{attribute 'qualified_only'}
{attribute 'strict'}
TYPE E_DALIBridgeCommand :
(
	idle,
	directArcPowerControl,
	queryActualLevel,
	queryStatus,
	setEventScheme,
	queryEventScheme,
	setEventFilter,
	queryEventFilter,
	identifyDevice102,
	identifyDevice103,
	enableInstance,
	goToScene,
	setFadeTime,
	queryInputValue,
	
	queryBatteryCharge,
	queryDurationTestResult,
	queryEmergencyMode,
	queryEmergencyStatus,
	queryFailureStatus,
	queryRatedDuration,
	queryTestTiming,
	resetDurationTestDoneFlag,
	resetFunctionTestDoneFlag,
	startDurationTest,
	startFunctionTest,
	stopTest,
	setDurationTestInterval,
	setFunctionTestInterval,
	startIdentification202,
	queryGroups,
	addToGroup,
	removeFromGroup,
	
	testCommand := 100
);
END_TYPE

(* stored: Version 1.1.0.1, ProductVersion 3.1.4024.11
   EnumerationTextList E_DALIBridgeCommand: Id {ace459ee-9ad7-4807-a32a-2eb1c3024f91} *)
